(* CODESYS project e!C_UnitConversion_Test_1.ecp

Project tree, tasks and I/O mapping:
  PFC200_CS_2ETH_RS : 750-8202 PFC200 2ETH RS, WAGO, order no. 0750-8202, version 5.11.1.16
    application PFC8202
      libraries: ; Unit Conversion Interfaces, * (Intern)
      task PLC_Task (cyclic, interval t#10ms, priority 14) calls PLC_PRG
      task VISU_TASK (cyclic, interval 100 ms, priority 15) calls VisuElems.Visu_Prg
      program PLC_PRG [ST]
      program POU_IO [ST]
      UnitConversion1
      visualisation Visu_Main
    DeviceAdapter
    Kbus : Kbus, WAGO, version 1.4.0.2
        unmapped channels: K-BUS diagnostics
      _8_DO_DI_Generic : 075x-8DO8DI, WAGO, order no. 075x-8DO8DI, version 0.0.0.13
          unmapped channels: _IN, _OUT
        DeviceAdapter
      _4_AO_4_20mA : 0750-0555, WAGO, order no. 0750-0555, version 0.0.0.12
          unmapped channels: _QW 1, _QW 2, _QW 3, _QW 4
        DeviceAdapter
      _4_AI_4_20mA_s_e : 0750-0455, WAGO, order no. 0750-0455, version 0.0.0.12
          unmapped channels: _IW 1, _IW 2, _IW 3, _IW 4
        DeviceAdapter
    MODBUS
      MODBUS : MODBUS, WAGO, order no. n/a, version 1.1.1.15
    Serial
      COM1 : COM1, WAGO, version 0.0.0.19
  libraries: WagoVisuIcons, 1.0.0.8 (WAGO)
  text list GlobalTextList
*)

// PFC200_CS_2ETH_RS/PFC8202/PLC_PRG
PROGRAM PLC_PRG
VAR
END_VAR


POU_IO();

END_PROGRAM

// PFC200_CS_2ETH_RS/PFC8202/POU_IO
PROGRAM POU_IO
VAR
	rTestVar1: REAL;
	rTestVar1_converted: REAL;
END_VAR



rTestVar1_converted := UnitConversionA.Convert(rValue:= rTestVar1);

END_PROGRAM

// PFC200_CS_2ETH_RS/PFC8202/Visu_Main
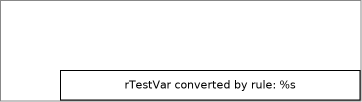
VISUALIZATION Visu_Main  // 362x102
    Rectangle (60,70 300x30), "rTestVar converted by rule: %s", text variable: POU_IO.rTestVar1
END_VISUALIZATION
